// Implicitly generated code : DO NOT EDIT
FUNCTION CheckPointer : POINTER TO BYTE
VAR_INPUT 
	ptToTest : POINTER TO BYTE; // Destination address of the pointer
	iSize : DINT;		        // Size of the type the pointer points to. (e.g: 20 for POINTER TO ARRAY [0..9] OF INT) 
	iGran : DINT;		        // Granularity of the pointer access. This is the size of the biggest non-structured data type in the type the pointer points to. (e.g: 2 for POINTER TO ARRAY [0..9] OF INT)
	bWrite: BOOL;		        // Indicates read or write Access. TRUE = write access.
END_VAR

// Implicitly generated code : Only an Implementation suggestion
{noflow}
IF ptToTest=0 THEN
    ADSLOGSTR(ADSLOG_MSGTYPE_ERROR OR ADSLOG_MSGTYPE_STRING,'CheckPointer failed due to invalid address.','');
ELSIF iSize<=0 THEN
    ADSLOGSTR(ADSLOG_MSGTYPE_ERROR OR ADSLOG_MSGTYPE_STRING,'CheckPointer failed due to invalid size.','');
ELSIF iGran<=0 THEN
    ADSLOGSTR(ADSLOG_MSGTYPE_ERROR OR ADSLOG_MSGTYPE_STRING,'CheckPointer failed due to invalid granularity.','');
// -> Please note that the following memory area check is time consuming:
//ELSIF F_CheckMemoryArea(pData:=ptToTest,nSize:=DINT_TO_UDINT(iSize)) = E_TcMemoryArea.Unknown THEN
//    ADSLOGSTR(ADSLOG_MSGTYPE_ERROR OR ADSLOG_MSGTYPE_STRING,'CheckPointer failed due to unknown memory area.','');
END_IF
CheckPointer := ptToTest;
{flow}

END_FUNCTION

(* stored: Version 1.1.0.1, ProductVersion 3.1.4024.12
   POU CheckPointer: Id {6c49341e-9c64-4f6c-9497-cc8b2e09a747}, SpecialFunc CheckPointer *)
